FUNCTION myFC : STRING
VAR_INPUT
	myInterface : ITF_MyTest;
END_VAR
VAR
END_VAR

myFC := myInterface.METH2();

END_FUNCTION

(* stored: Version 1.1.0.1, ProductVersion 3.1.4024.12
   POU myFC: Id {659586f2-b418-4108-afc0-bf786f6d3078}, SpecialFunc None *)
